// CALCULATE CURRENT REACTION RATE [mol/m3/s]

FUNCTION GetReactRate : REAL

VAR
	
	// Module A [(mol/m3)2]
	a : REAL := EXPT(Conc.now,2); 
	
	// Module B [m3/mol/s]
	b : REAL := Const.Rk; 
	
	// Module C []
	kelvin : REAL := temp.now + temp.offset;
	AE     : REAL := const.AE;
	c      : REAL;
	
END_VAR

// Error handling
IF kelvin <= 0 THEN
	getreactrate :=0;
	RETURN;
END_IF

c := EXP(-AE / kelvin);

// [mol2/m32 * m3/mol/s -> mol/m3/s]
GetReactRate := a * b * c;

END_FUNCTION

(* stored: Version 1.1.0.1, ProductVersion 3.1.4024.12
   POU GetReactRate: Id {ac67f14b-de86-4e0f-b024-f80724755f36}, SpecialFunc None *)
